// TIA Portal V17 export
// export: Created 2024-09-02T12:50:15.1853297Z, ExportSetting WithDefaults, DisplayName Totally Integrated Automation Portal, DisplayVersion V17, DisplayName TIA Portal Openness, DisplayVersion V17, DisplayName TIA Portal Version Control Interface, DisplayVersion V17, DisplayName STEP 7 Professional, DisplayVersion V17, DisplayName STEP 7 Safety, DisplayVersion V17, DisplayName WinCC Professional, DisplayVersion V17
FUNCTION "AnwFC_ZP_door_OP70" : Void   // FC149, LAD
TITLE = Safety door / Schutztüren
{ S7_Optimized_Access := 'TRUE' }
AUTHOR : OlegFuehrus
FAMILY : SG
NAME : SG
VERSION : 0.1
// stored: AutoNumber true, IsIECCheckEnabled false, SetENOAutomatically false, UDAEnableTagReadback false
   VAR_TEMP
      Enable_Opening : Bool;
   END_VAR
   VAR_TEMP   // added for the SCL form of the ladder/FBD networks
      _w1 : Bool;
   END_VAR
BEGIN

REGION Network 1: Protective doors: stop cycle end / Schutztüren: Halt Takt Ende
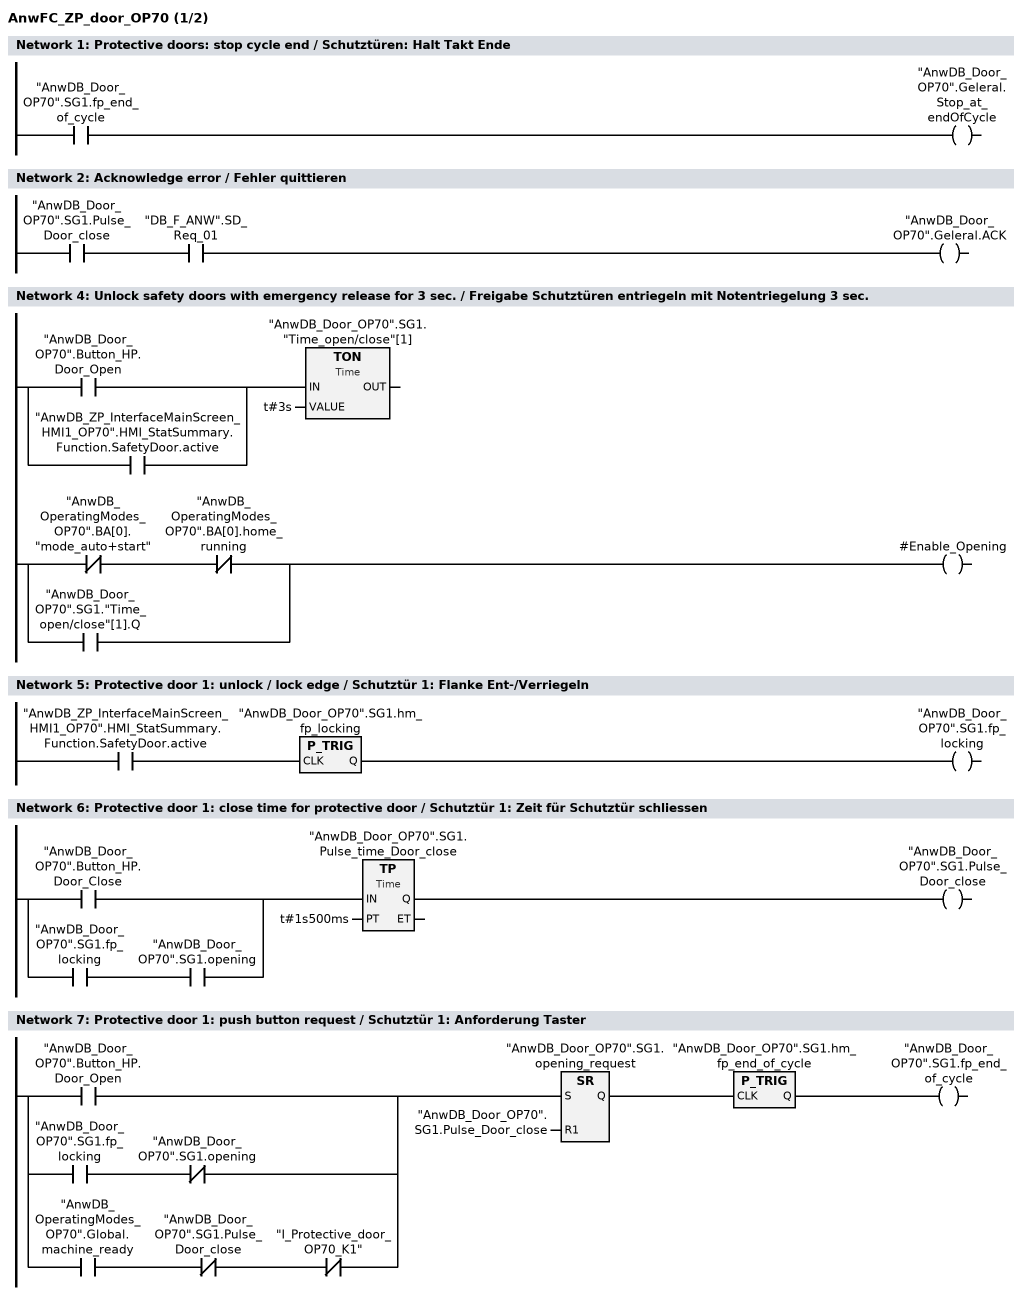
   RUNG wire#powerrail
      Contact( "AnwDB_Door_OP70".SG1.fp_end_of_cycle )
      Coil( "AnwDB_Door_OP70".Geleral.Stop_at_endOfCycle )
   END_RUNG
   // the same network as SCL:
   "AnwDB_Door_OP70".Geleral.Stop_at_endOfCycle := "AnwDB_Door_OP70".SG1.fp_end_of_cycle;
END_REGION

REGION Network 2: Acknowledge error / Fehler quittieren
   RUNG wire#powerrail
      Contact( "AnwDB_Door_OP70".SG1.Pulse_Door_close )
      Contact( "DB_F_ANW".SD_Req_01 )
      Coil( "AnwDB_Door_OP70".Geleral.ACK )
   END_RUNG
   // the same network as SCL:
   "AnwDB_Door_OP70".Geleral.ACK := "AnwDB_Door_OP70".SG1.Pulse_Door_close AND "DB_F_ANW".SD_Req_01;
END_REGION

REGION Network 3: ----------------------------------- Safety Door 1 -------------------------------------- / ----------------------------------- Schutztür 1 --------------------------------------
END_REGION

REGION Network 4: Unlock safety doors with emergency release for 3 sec. / Freigabe Schutztüren entriegeln mit Notentriegelung 3 sec.
   "AnwDB_Door_OP70".SG1."Time_open/close"[1].TON(IN := "AnwDB_Door_OP70".Button_HP.Door_Open OR "AnwDB_ZP_InterfaceMainScreen_HMI1_OP70".HMI_StatSummary.Function.SafetyDoor.active, PT := t#3s);   // TON coil
   #Enable_Opening := (NOT "AnwDB_OperatingModes_OP70".BA[0]."mode_auto+start" AND NOT "AnwDB_OperatingModes_OP70".BA[0].home_running) OR "AnwDB_Door_OP70".SG1."Time_open/close"[1].Q;
END_REGION

REGION Network 5: Protective door 1: unlock / lock edge / Schutztür 1: Flanke Ent-/Verriegeln
   RUNG wire#powerrail
      Contact( "AnwDB_ZP_InterfaceMainScreen_HMI1_OP70".HMI_StatSummary.Function.SafetyDoor.active )
      P_Trig( "AnwDB_Door_OP70".SG1.hm_fp_locking )
      Coil( "AnwDB_Door_OP70".SG1.fp_locking )
   END_RUNG
   // the same network as SCL:
   #_w1 := "AnwDB_ZP_InterfaceMainScreen_HMI1_OP70".HMI_StatSummary.Function.SafetyDoor.active AND NOT "AnwDB_Door_OP70".SG1.hm_fp_locking;   // rising edge
   "AnwDB_Door_OP70".SG1.hm_fp_locking := "AnwDB_ZP_InterfaceMainScreen_HMI1_OP70".HMI_StatSummary.Function.SafetyDoor.active;
   "AnwDB_Door_OP70".SG1.fp_locking := #_w1;
END_REGION

REGION Network 6: Protective door 1: close time for protective door / Schutztür 1: Zeit für Schutztür schliessen
   RUNG wire#powerrail
      Contact( "AnwDB_Door_OP70".Button_HP.Door_Close )
      wire#w1
      { S7_Templates := "time_type := Time" } "AnwDB_Door_OP70".SG1.Pulse_time_Door_close.TP(pt := t#1s500ms, et =>)
      Coil( "AnwDB_Door_OP70".SG1.Pulse_Door_close )
   END_RUNG
   RUNG wire#powerrail
      Contact( "AnwDB_Door_OP70".SG1.fp_locking )
      Contact( "AnwDB_Door_OP70".SG1.opening )
   END_RUNG wire#w1
   // the same network as SCL:
   "AnwDB_Door_OP70".SG1.Pulse_time_Door_close.TP(IN := "AnwDB_Door_OP70".Button_HP.Door_Close OR ("AnwDB_Door_OP70".SG1.fp_locking AND "AnwDB_Door_OP70".SG1.opening),
                           PT := t#1s500ms);
   "AnwDB_Door_OP70".SG1.Pulse_Door_close := "AnwDB_Door_OP70".SG1.Pulse_time_Door_close.Q;
END_REGION

REGION Network 7: Protective door 1: push button request / Schutztür 1: Anforderung Taster
   RUNG wire#powerrail
      Contact( "AnwDB_Door_OP70".Button_HP.Door_Open )
      wire#w1
      S_SR(operand := "AnwDB_Door_OP70".SG1.opening_request, r1 := "AnwDB_Door_OP70".SG1.Pulse_Door_close)
      P_Trig( "AnwDB_Door_OP70".SG1.hm_fp_end_of_cycle )
      Coil( "AnwDB_Door_OP70".SG1.fp_end_of_cycle )
   END_RUNG
   RUNG wire#powerrail
      Contact( "AnwDB_Door_OP70".SG1.fp_locking )
      I_Contact( "AnwDB_Door_OP70".SG1.opening )
   END_RUNG wire#w1
   RUNG wire#powerrail
      Contact( "AnwDB_OperatingModes_OP70".Global.machine_ready )
      I_Contact( "AnwDB_Door_OP70".SG1.Pulse_Door_close )
      I_Contact( "I_Protective_door_OP70_K1" )
   END_RUNG wire#w1
   // the same network as SCL:
   IF "AnwDB_Door_OP70".Button_HP.Door_Open OR ("AnwDB_Door_OP70".SG1.fp_locking AND NOT "AnwDB_Door_OP70".SG1.opening) OR ("AnwDB_OperatingModes_OP70".Global.machine_ready AND NOT "AnwDB_Door_OP70".SG1.Pulse_Door_close AND NOT "I_Protective_door_OP70_K1") THEN
       "AnwDB_Door_OP70".SG1.opening_request := TRUE;   // SR flip-flop
   END_IF;
   IF "AnwDB_Door_OP70".SG1.Pulse_Door_close THEN "AnwDB_Door_OP70".SG1.opening_request := FALSE; END_IF;
   #_w1 := "AnwDB_Door_OP70".SG1.opening_request AND NOT "AnwDB_Door_OP70".SG1.hm_fp_end_of_cycle;   // rising edge
   "AnwDB_Door_OP70".SG1.hm_fp_end_of_cycle := "AnwDB_Door_OP70".SG1.opening_request;
   "AnwDB_Door_OP70".SG1.fp_end_of_cycle := #_w1;
END_REGION

REGION Network 8: Protective door 1: unlock / Schutztür 1: entriegeln
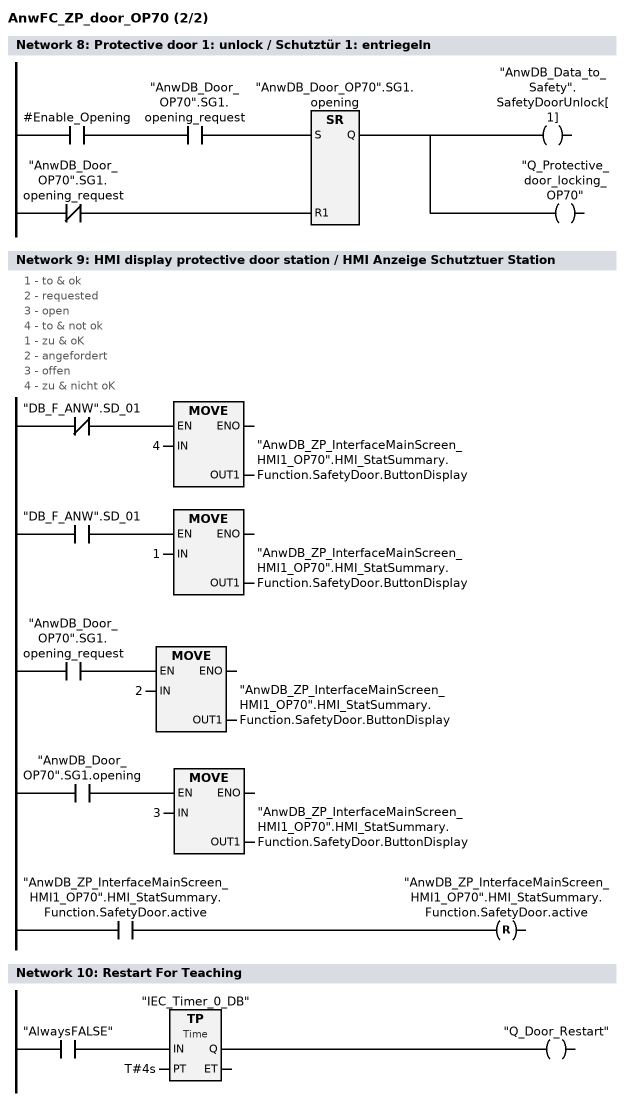
   RUNG wire#powerrail
      Contact( #Enable_Opening )
      Contact( "AnwDB_Door_OP70".SG1.opening_request )
      S_SR(operand := "AnwDB_Door_OP70".SG1.opening, r1 := wire#w1)
      wire#w2
      Coil( "AnwDB_Data_to_Safety".SafetyDoorUnlock[1] )
   END_RUNG
   RUNG wire#powerrail
      I_Contact( "AnwDB_Door_OP70".SG1.opening_request )
   END_RUNG wire#w1
   RUNG wire#w2
      Coil( "Q_Protective_door_locking_OP70" )
   END_RUNG
   // the same network as SCL:
   IF #Enable_Opening AND "AnwDB_Door_OP70".SG1.opening_request THEN
       "AnwDB_Door_OP70".SG1.opening := TRUE;   // SR flip-flop
   END_IF;
   IF NOT "AnwDB_Door_OP70".SG1.opening_request THEN "AnwDB_Door_OP70".SG1.opening := FALSE; END_IF;
   "AnwDB_Data_to_Safety".SafetyDoorUnlock[1] := "AnwDB_Door_OP70".SG1.opening;
   "Q_Protective_door_locking_OP70" := "AnwDB_Door_OP70".SG1.opening;
END_REGION

REGION Network 9: HMI display protective door station / HMI Anzeige Schutztuer Station
   // 1 - to & ok
   // 2 - requested
   // 3 - open
   // 4 - to & not ok
   // 1 - zu & oK
   // 2 - angefordert
   // 3 - offen
   // 4 - zu & nicht oK
   RUNG wire#powerrail
      I_Contact( "DB_F_ANW".SD_01 )
      Move(in := 4, out1 => "AnwDB_ZP_InterfaceMainScreen_HMI1_OP70".HMI_StatSummary.Function.SafetyDoor.ButtonDisplay)
   END_RUNG
   RUNG wire#powerrail
      Contact( "DB_F_ANW".SD_01 )
      Move(in := 1, out1 => "AnwDB_ZP_InterfaceMainScreen_HMI1_OP70".HMI_StatSummary.Function.SafetyDoor.ButtonDisplay)
   END_RUNG
   RUNG wire#powerrail
      Contact( "AnwDB_Door_OP70".SG1.opening_request )
      Move(in := 2, out1 => "AnwDB_ZP_InterfaceMainScreen_HMI1_OP70".HMI_StatSummary.Function.SafetyDoor.ButtonDisplay)
   END_RUNG
   RUNG wire#powerrail
      Contact( "AnwDB_Door_OP70".SG1.opening )
      Move(in := 3, out1 => "AnwDB_ZP_InterfaceMainScreen_HMI1_OP70".HMI_StatSummary.Function.SafetyDoor.ButtonDisplay)
   END_RUNG
   RUNG wire#powerrail
      Contact( "AnwDB_ZP_InterfaceMainScreen_HMI1_OP70".HMI_StatSummary.Function.SafetyDoor.active )
      R_Coil( "AnwDB_ZP_InterfaceMainScreen_HMI1_OP70".HMI_StatSummary.Function.SafetyDoor.active )
   END_RUNG
   // the same network as SCL:
   IF NOT "DB_F_ANW".SD_01 THEN
       "AnwDB_ZP_InterfaceMainScreen_HMI1_OP70".HMI_StatSummary.Function.SafetyDoor.ButtonDisplay := 4;
   END_IF;
   IF "DB_F_ANW".SD_01 THEN
       "AnwDB_ZP_InterfaceMainScreen_HMI1_OP70".HMI_StatSummary.Function.SafetyDoor.ButtonDisplay := 1;
   END_IF;
   IF "AnwDB_Door_OP70".SG1.opening_request THEN
       "AnwDB_ZP_InterfaceMainScreen_HMI1_OP70".HMI_StatSummary.Function.SafetyDoor.ButtonDisplay := 2;
   END_IF;
   IF "AnwDB_Door_OP70".SG1.opening THEN
       "AnwDB_ZP_InterfaceMainScreen_HMI1_OP70".HMI_StatSummary.Function.SafetyDoor.ButtonDisplay := 3;
   END_IF;
   IF "AnwDB_ZP_InterfaceMainScreen_HMI1_OP70".HMI_StatSummary.Function.SafetyDoor.active THEN
       "AnwDB_ZP_InterfaceMainScreen_HMI1_OP70".HMI_StatSummary.Function.SafetyDoor.active := FALSE;
   END_IF;
END_REGION

REGION Network 10: Restart For Teaching
   RUNG wire#powerrail
      Contact( "AlwaysFALSE" )
      { S7_Templates := "time_type := Time" } "IEC_Timer_0_DB".TP(pt := T#4s, et =>)
      Coil( "Q_Door_Restart" )
   END_RUNG
   // the same network as SCL:
   "IEC_Timer_0_DB".TP(IN := "AlwaysFALSE", PT := T#4s);
   "Q_Door_Restart" := "IEC_Timer_0_DB".Q;
END_REGION

REGION Network 11: END
END_REGION
END_FUNCTION
